ABB RAPID module: Wobj_wobj_Pick.mod

MODULE Wobj_wobj_Pick
	! Points are read in order of declaration.
  ! Please do not change the order of points!

  LOCAL PERS robtarget pWobj_U_PointX1:=[[-730.5011,2011.136,-53.266],[0.695277631282806,-0.718628406524658,-0.00798139721155167,0.00992555543780327],[1,-2,0,0],[0,9E+09,9E+09,9E+09,9E+09,9E+09]];
	LOCAL PERS robtarget pWobj_U_PointX2:=[[-1150.647,1999.545,-48.36156],[0.695280075073242,-0.718623578548431,-0.00806344021111727,0.0100353769958019],[1,-2,0,0],[0,9E+09,9E+09,9E+09,9E+09,9E+09]];
	LOCAL PERS robtarget pWobj_U_PointY1:=[[-1130.292,1461.221,-55.50463],[0.695284724235535,-0.718619048595428,-0.00806234683841467,0.0100415125489235],[1,-2,0,0],[0,9E+09,9E+09,9E+09,9E+09,9E+09]];

ENDMODULE
